{attribute addProperty BoxType "EL3751-0000-0020"}
{attribute addProperty Id "StatusAT %I*Status_6A40DED4324"}
{attribute addProperty CRC "3480367792"}
{attribute addProperty SizeInBites "32"}
{attribute addProperty SizeInBytes "4"}
TYPE PAI_Status_CF7232B0 :
STRUCT
	{attribute addProperty Name "Status"}
	Status AT %I* : Status_6A40DED4;
END_STRUCT
END_TYPE

(* stored: Version 1.2.0.0, ProductVersion 3.1.4024.9
   DUT PAI_Status_CF7232B0: Id {0b47d179-3a31-4abc-8007-4e73f7151792} *)
